FUNCTION_BLOCK E_F_DIV (* Event-Driven Frequency Divider *)
  (* Standard: 61499-2 *)
  (* Version 0.0, 2004-04-23, JHC, Rockwell Automation *)
  (* Compiler header: package fb.rt.events; *)
  (* Compiler Java Sun JDK 1.06 *)
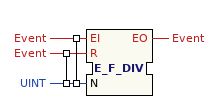
  EVENT_INPUT
    EI WITH N; (* Input Event *)
    R WITH N; (* Reset Divider *)
  END_EVENT
  EVENT_OUTPUT
    EO; (* Output Event at frequency 1/N of EI *)
  END_EVENT
  VAR_INPUT
    N : UINT := 1; (* Divisor (should be >0) *)
  END_VAR
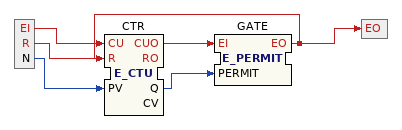
  FBS
    CTR : E_CTU;
    GATE : E_PERMIT;
  END_FBS
  EVENT_CONNECTIONS
    R TO CTR.R;
    EI TO CTR.CU;
    CTR.CUO TO GATE.EI;
    GATE.EO TO CTR.R;
    GATE.EO TO EO;
  END_CONNECTIONS
  DATA_CONNECTIONS
    N TO CTR.PV;
    CTR.Q TO GATE.PERMIT;
  END_CONNECTIONS
END_FUNCTION_BLOCK
